Staubli VAL3: selectItem.pgx

public program selectItem(num x_nIndex)
  local InstrItem l_sItem
begin
  //
  // select or unselect one item
  //
  call getItem(l_sItem,x_nIndex)
  if find(l_sItem.sType,"#")==-1
    l_sItem.sType="#"+l_sItem.sType
  else
    l_sItem.sType=right(l_sItem.sType,len(l_sItem.sType)-1)
  endIf
  // set Item
  call setItem(l_sItem,x_nIndex)
end
